ABB RobotStudio station: plantilla - pruebas_20220202-184230.rsstn

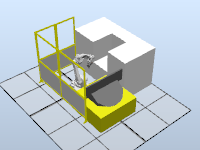
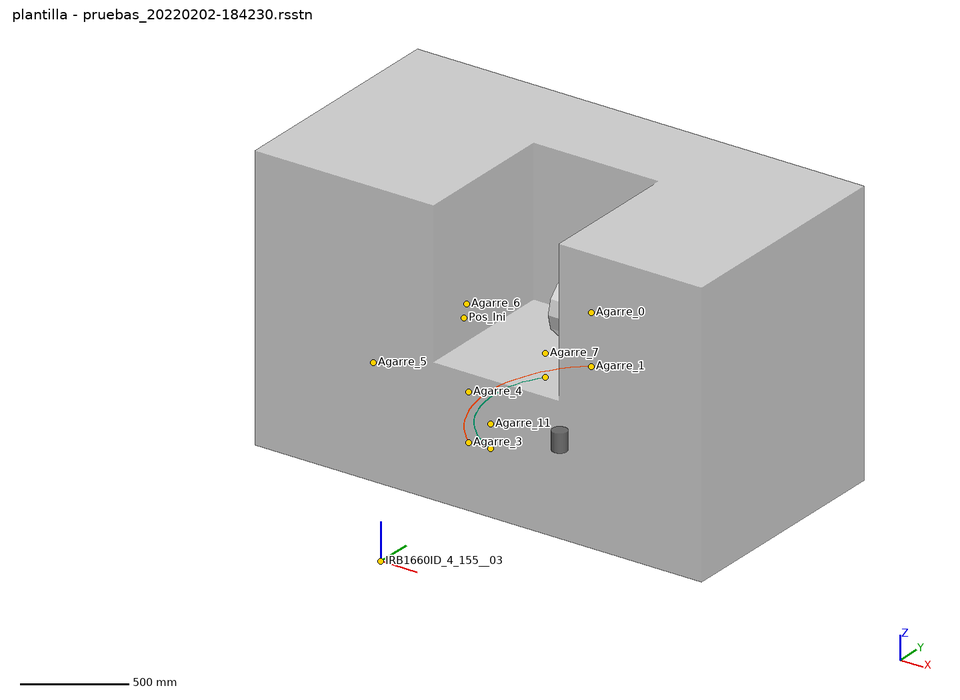
[picture v1: parts stored in the station drawn from their meshes, with robot base, taught points and paths (robot models come from the ABB library and are not in the file)]
Station Station (saved by RobotStudio 21.2.9526.0)
Controller Controlador2_Porta
  mechanical unit ROB_1: IRB1660ID_4_155__03, 6 joints, base frame (0, 0, 0) mm
  mechanical unit Portapiezas: Portapiezas, 2 joints, base frame (1275, -81, 0) mm, rotated rx 0 ry 0 rz 176.36 deg
Layout (positions relative to the parent item):
  - IRB1660ID_4_155__03 [mechanism, from Robots\IRB1660ID_4_155__03.rslib] at (0, 0, 0) mm; joint values [0.0253, -0.3978, -0.0059, 0.0191, 1.9827, 1.1981] (rad or m)
  - Pinza_1 [mechanism, from Efectores_finales - Copy\PinzaF_1.rslib] at (457.74, 13.95, 1364.34) mm, rotated rx -179.93 ry -1.11 rz 113.24 deg; joint values [0, 0] (rad or m)
  - Pinza_2 [mechanism, from Efectores_finales - Copy\PinzaF_2.rslib] at (457.74, 13.95, 1364.34) mm, rotated rx -179.93 ry -1.11 rz 113.24 deg; joint values [0, 0] (rad or m)
  - Torno [part] at (-1172.42, 1966.27, 0) mm, rotated rx 0 ry 0 rz 180 deg, size 2500 x 1300 x 1500 mm
  - Fence_740 [graphiccomponentgroup, from Equipment\Fence_740.rslib] at (-1160.76, -802.49, 0) mm
    - Body 1 [part, from Equipment\Fence_740.rslib]
    - Body 2 [part, from Equipment\Fence_740.rslib]
  - Fence_2500 [graphiccomponentgroup, from Equipment\Fence_2500.rslib] at (1297.15, -826.85, 0) mm, rotated rx 0 ry 0 rz 90 deg
    - Body 1 [part, from Equipment\Fence_2500.rslib]
    - Body 2 [part, from Equipment\Fence_2500.rslib]
  - Fence_740_2 [graphiccomponentgroup, from Equipment\Fence_740.rslib] at (-1148.66, -57.63, 0) mm
    - Body 1 [part, from Equipment\Fence_740.rslib]
    - Body 2 [part, from Equipment\Fence_740.rslib]
  - Portapiezas [mechanism] at (0, 0, 0) mm; joint values [0, 0] (rad or m)
      links: L1, L2, L3
  - Cilindros [part] at (500, -500, 850) mm, size 80 x 79.4 x 100 mm
Attachment: Pinza_1 is attached to IRB1660ID_4_155__03 / Link6
Attachment: Pinza_2 is attached to IRB1660ID_4_155__03 / Link6
Attachment: Cilindros is attached to Portapiezas / L3
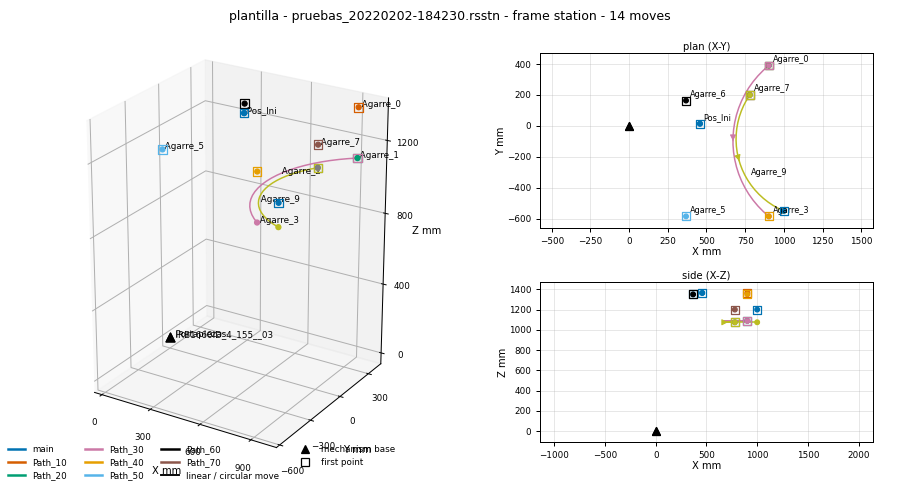
[picture p0: tool path of plantilla - pruebas_20220202-184230.rsstn in frame station, 14 of 14 moves have a stored position in this frame; points joined in program order, loops and branches not executed]
Targets, tools, work objects and paths stored in the station, written as RAPID:
! task T_ROB1
MODULE CalibData
  PERS tooldata Pinza_1:=[TRUE,[[-100,0,70],[0.707106781,0,-0.707106781,0]],[1,[0,0,1],[1,0,0,0],0,0,0]];
  PERS tooldata Vara:=[TRUE,[[0,0,250],[0.707106781,0,0,0.707106781]],[1,[0,0,1],[1,0,0,0],0,0,0]];
  PERS tooldata Soplador:=[TRUE,[[0,-70,70],[0.5,0.5,-0.5,0.5]],[1,[0,0,1],[1,0,0,0],0,0,0]];
  PERS tooldata Pinza_2_1:=[TRUE,[[100,0,70],[0.707106781,0,0.707106781,0]],[1,[0,0,2],[1,0,0,0],0,0,0]];
ENDMODULE

! task T_ROB1
MODULE Module1
  CONST robtarget Agarre_1:=[[902.905242443,390.185715306,1089.467071419],[0.008413664,-0.550176032,-0.8349924,-0.004820384],[0,0,0,0],[0,0,9E+09,9E+09,9E+09,9E+09]];
  CONST robtarget Agarre_0:=[[902.905238891,390.185714028,1364.343070082],[0.008413683,-0.550176024,-0.834992405,-0.004820355],[0,0,1,0],[0,0,9E+09,9E+09,9E+09,9E+09]];
  CONST robtarget Pos_Ini:=[[457.741499845,13.951470202,1364.343080589],[0.008413673,-0.550176028,-0.834992403,-0.004820372],[0,0,0,0],[0,0,9E+09,9E+09,9E+09,9E+09]];
  CONST robtarget Agarre_3:=[[902.905225,-584.982599934,1089.467084686],[0.008413653,-0.550176031,-0.834992401,-0.004820384],[-1,0,0,0],[90,0,9E+09,9E+09,9E+09,9E+09]];
  CONST robtarget Agarre_2:=[[677.219996128,-8.495218742,1089.467073949],[0.008413714,-0.550176032,-0.8349924,-0.004820352],[-1,0,0,0],[45,0,9E+09,9E+09,9E+09,9E+09]];
  CONST robtarget Agarre_4:=[[902.905215745,-584.982593979,1350.189011707],[0.008413694,-0.550176033,-0.834992399,-0.004820384],[-1,0,0,0],[90.000002504,0,9E+09,9E+09,9E+09,9E+09]];
  CONST robtarget Agarre_5:=[[367.553891268,-584.982601827,1350.188994453],[0.008413681,-0.550176029,-0.834992402,-0.004820378],[-1,0,0,0],[90.000002504,0,9E+09,9E+09,9E+09,9E+09]];
  CONST robtarget Agarre_6:=[[367.553892033,163.63039142,1350.189002852],[0.008413628,-0.550176005,-0.834992418,-0.004820404],[0,0,1,0],[90.000002504,0,9E+09,9E+09,9E+09,9E+09]];
  CONST robtarget Agarre_8:=[[779.999980593,200.000005322,1075.000071425],[0.008424643,-0.550158387,-0.835003922,-0.004819277],[0,0,0,0],[90,0,9E+09,9E+09,9E+09,9E+09]];
  CONST robtarget Agarre_7:=[[779.999991418,200.000007857,1200.000072424],[0.008424613,-0.550158412,-0.835003905,-0.004819308],[0,0,0,0],[90.000002504,0,9E+09,9E+09,9E+09,9E+09]];
  CONST robtarget Agarre_9:=[[760.000001353,-340.000005904,1075.000071669],[0.008424643,-0.550158378,-0.835003927,-0.004819292],[-1,0,0,0],[145,0,9E+09,9E+09,9E+09,9E+09]];
  CONST robtarget Agarre_10:=[[1000.000037283,-550.000003833,1075.00006573],[0.008424622,-0.550158381,-0.835003926,-0.004819294],[-1,0,0,0],[180,0,9E+09,9E+09,9E+09,9E+09]];
  CONST robtarget Agarre_11:=[[1000.000038498,-550.000004351,1200.000062962],[0.008424624,-0.550158384,-0.835003924,-0.004819294],[-1,0,0,0],[180.000005009,0,9E+09,9E+09,9E+09,9E+09]];
  CONST robtarget Pos_Final:=[[457.74150017,13.95147021,1364.34307978],[0.008413673,-0.550176028,-0.834992403,-0.004820372],[0,0,0,0],[180,0,9E+09,9E+09,9E+09,9E+09]];
  PROC main()
    MoveL Pos_Ini,v300,fine,tool0\WObj:=wobj0;
    Path_10;
    Path_20;
    Path_30;
    Path_40;
    Path_50;
    Path_60;
    Path_70;
    Path_70;
    Path_80;
    Path_90;
    Path_100;
    MoveL Pos_Final,v300,fine,tool0\WObj:=wobj0;
  ENDPROC
  PROC Path_10()
    MoveL Agarre_0,v300,fine,tool0\WObj:=wobj0;
  ENDPROC
  PROC Path_20()
    MoveL Agarre_1,v300,fine,tool0\WObj:=wobj0;
  ENDPROC
  PROC Path_30()
    MoveL Agarre_1,v300,fine,tool0\WObj:=wobj0;
    MoveC Agarre_2,Agarre_3,v300,fine,tool0\WObj:=wobj0;
  ENDPROC
  PROC Path_40()
    MoveL Agarre_4,v300,fine,tool0\WObj:=wobj0;
  ENDPROC
  PROC Path_50()
    MoveL Agarre_5,v300,fine,tool0\WObj:=wobj0;
  ENDPROC
  PROC Path_60()
    MoveL Agarre_6,v300,fine,tool0\WObj:=wobj0;
  ENDPROC
  PROC Path_70()
    MoveL Agarre_7,v300,fine,tool0\WObj:=wobj0;
  ENDPROC
  PROC Path_80()
    MoveL Agarre_8,v300,fine,tool0\WObj:=wobj0;
  ENDPROC
  PROC Path_90()
    MoveL Agarre_8,v300,fine,tool0\WObj:=wobj0;
    MoveC Agarre_9,Agarre_10,v300,fine,tool0\WObj:=wobj0;
  ENDPROC
  PROC Path_100()
    MoveL Agarre_11,v300,fine,tool0\WObj:=wobj0;
  ENDPROC
ENDMODULE

